PROGRAM MAIN
VAR
	nCounter : INT ;
END_VAR

nCounter := nCounter + 1;

END_PROGRAM

(* stored: Version 1.1.0.1, ProductVersion 3.1.4024.12
   POU MAIN: Id {bb779d4c-6bb8-4ba4-9107-b801c363bbec}, SpecialFunc None *)
